PROGRAM MAIN
VAR CONSTANT
	//Constants to set maximum matrix size at compile time
	cMaxRows:INT:=4;
	cMaxCols:INT:=3;
END_VAR
VAR
	//Configure Dispense Matrix [4,3]
	fbDispenseMatrix:FB_Matrix;
	aDispenseMatrixConfig : ARRAY [1..cMaxRows,1..cMaxCols] OF ST_SolenoidConfig;
	bDispMatrixEnable:BOOL;
	bDispMatrixReset:BOOL;
	Disp_st_path : ST_Path;
	bDispFindPath: BOOL;
	bDispPathingSwitch:BOOL;
	nDispenseRows:INT:=4;
	nDispenseCols:INT:=3;
	
	//Configure Inlet Matrix [2,3]
	fbInletMatrix:FB_Matrix;
	aInletMatrixConfig: ARRAY [1..cMaxRows,1..cMaxCols] OF ST_SolenoidConfig;
	bInletMatrixEnable:BOOL;
	bInletMatrixReset:BOOL;
	Inlet_st_path : ST_Path;
	bInletFindPath: BOOL;
	bInletPathingSwitch:BOOL;
	nInletRows:INT:=2;
	nInletCols:INT:=3;
	
	//Configure Filling Matrix [4,3]
	fbFillMatrix:FB_Matrix;
	aFillMatrixConfig : ARRAY [1..cMaxRows,1..cMaxCols] OF ST_SolenoidConfig;
	bFillMatrixEnable:BOOL;
	bFillMatrixReset:BOOL;
	Fill_st_path : ST_Path;
	bFillFindPath: BOOL;
	bFillPathingSwitch:BOOL;
	nFillRows:INT:=4;
	nFillCols:INT:=3;	
	
	//Array of Pressure Transducers
	aPT: ARRAY [1.. GVL_IO.cNumofPT] OF FB_PressureTransducer;
	
	//Standard Config Parameter Struct for Pressure and Temp sensors
	stAnalogCfg : ST_AnalogPressureTemp;
	
	//Initialising Boolean 
	bInitialise:BOOL:=TRUE;
END_VAR

//Run Initialise Method once on first cycle
IF bInitialise THEN
	M_Initalize();
	bInitialise:=FALSE;
END_IF

//Update sensors from IO
M_Sensors();

//Calling FB_MAtrix for each of the three matrices of valves, Dispense, Inlet and FIlling.
fbDispenseMatrix(bDeviceEnable:=bDispMatrixEnable,bDeviceReset:=bDispMatrixReset,
	            aConfig:=aDispenseMatrixConfig,st_path:=Disp_st_path,bSetCurrentPath:=bDispFindPath,
                bPathingOn:=bDispPathingSwitch,nRowSize:=nDispenseRows,nColSize:=nDispenseCols);
				
fbInletMatrix(bDeviceEnable:=bInletMatrixEnable,bDeviceReset:=bInletMatrixReset,aConfig:=aInletMatrixConfig,
	          st_path:=Inlet_st_path,bSetCurrentPath:=bInletFindPath,bPathingOn:=bInletPathingSwitch,
			  nRowSize:=nInletRows,nColSize:=nInletCols);
			  
fbFillMatrix(bDeviceEnable:=bFillMatrixEnable,bDeviceReset:=bFillMatrixReset,aConfig:=aFillMatrixConfig,
	          st_path:=Fill_st_path,bSetCurrentPath:=bFillFindPath,bPathingOn:=bFillPathingSwitch,
			  nRowSize:=nFillRows,nColSize:=nFillCols);

				
//Update the inputs to the matrix functions and pressure sensors from GVLs
M_UpdateFromHMI();

METHOD M_ActuateValves
VAR_INPUT
	rows:INT;
	cols:INT;
END_VAR
END_METHOD

METHOD PUBLIC M_Initalize 
VAR
rows:INT;
cols:INT;
END_VAR

//Configure the pressure sensors
	stAnalogCfg.rWarninglevel:=500;
	stAnalogCfg.rErrorLevel:=525;
	stAnalogCfg.rPressureMinSP:=0;
	stAnalogCfg.rPressureMaxSP:=1000;
	stAnalogCfg.rTemperatureMinSP:=-40;
	stAnalogCfg.rTemperatureMaxSP:=125;
	stAnalogCfg.nRawMin:=0;
	stAnalogCfg.nRawMax:=32767;
//Configure the pressure sensors
FOR rows:=1 TO GVL_IO.cNumofPT DO
    aPT[rows].st_AnalogPressureTempdata:=stAnalogCfg;
	apT[rows].sTag:=GVL_IO.sPTTags[rows];
END_FOR


//Initialise all matrices to be NC and to be un-energised
    FOR  rows:=1 TO cMaxRows DO
       FOR  cols:=1 TO cMaxCols DO
          aDispenseMatrixConfig[rows,cols].NormallyOpen:=FALSE;
		  aInletMatrixConfig[rows,cols].NormallyOpen:=FALSE;
		  aDispenseMatrixConfig[rows,cols].bOpen:=FALSE;
		  aInletMatrixConfig[rows,cols].bOpen:=FALSE;
		  aFillMatrixConfig[rows,cols].NormallyOpen:=FALSE;
		  aFillMatrixConfig[rows,cols].bOpen:=FALSE;
       END_FOR
    END_FOR
END_METHOD

METHOD M_Sensors
VAR
	nsensorNumber:INT;
END_VAR
FOR nsensorNumber:=1 TO GVL_IO.cNumofPT DO
	aPT[nsensorNumber](bDeviceEnable:=GVL_HMI.bEnableSensors,
		               bDeviceReset:=GVL_HMI.bResetSensors,
					   nSensorPressure:=GVL_IO.aPressRaw[nsensorNumber],
					   nSensorTemperature:=GVL_IO.aTempRaw[nsensorNumber],
					   rEngPressure=>GVL_HMI.aPV[nsensorNumber],
					   rEngTemperature=>GVL_HMI.aTV[nsensorNumber],
                       eDeviceState=>GVL_HMI.aSensorErrors[nsensorNumber]);			   
END_FOR
END_METHOD

METHOD M_UpdateDispenseFromHMI
VAR
	rows:INT;
	cols:INT;
END_VAR
//Variables for actuating the Dispense matrix updated from GVL here
bDispMatrixEnable:=GVL_HMI.bDispTurnOnMatrix;
bDispMatrixReset:=GVL_HMI.bDispResetMatrix;
Disp_st_path.endPath:=GVL_HMI.eDispEndOfPath;
Disp_st_path.startPath:=GVL_HMI.eDispStartOfPath;
bDispFindPath:=GVL_HMI.bDispActuatePath;
bDispPathingSwitch:=GVL_HMI.bDispTurnOnPathing;

//Change the display state of the matrix valves on the HMI screen
GVL_HMI.aDispStateofValves:=fbDispenseMatrix.aValveStates;

//Condition to avoid manual control when pathing is on
IF GVL_HMI.bDispTurnOnPathing THEN
	RETURN;
END_IF
FOR rows := 1 TO nDispenseRows DO
       FOR cols := 1 TO nDispenseCols DO
          aDispenseMatrixConfig[rows,cols].bOpen:=GVL_HMI.aDispManualValveSelection[rows,cols];
       END_FOR
END_FOR
END_METHOD

METHOD M_UpdateFillFromHMI
VAR
	rows:INT;
	cols:INT;
END_VAR
//Variables for actuating the filling matrix are updated from GVL here
bFillMatrixEnable:=GVL_HMI.bFillTurnOnMatrix;
bFillMatrixReset:=GVL_HMI.bFillResetMatrix;
bFillFindPath:=GVL_HMI.bFillActuatePath;
bFillPathingSwitch:=GVL_HMI.bFillTurnOnPathing;
Fill_st_path.endPath:=GVL_HMI.eFillEndOfPath;
Fill_st_path.startPath:=GVL_HMI.eFillStartOfPath;

//Change the display state of the matrix valves on the HMI screen
GVL_HMI.aFillStateofValves:=fbFillMatrix.aValveStates;


//Condition to avoid manual control when pathing is on
IF GVL_HMI.bFillTurnOnPathing THEN
	RETURN;
END_IF
FOR rows := 1 TO nFillRows DO
       FOR cols := 1 TO nFillCols DO
          aFillMatrixConfig[rows,cols].bOpen:=GVL_HMI.aFillManualValveSelection[rows,cols];
       END_FOR
END_FOR
END_METHOD

METHOD M_UpdateFromHMI
//Update each matrix Independently
M_UpdateDispenseFromHMI();
M_UpdateInletFromHMI();
M_UpdateFillFromHMI();
END_METHOD

METHOD M_UpdateInletFromHMI
VAR
	rows:INT;
	cols:INT;
END_VAR
//Variables for actuating the inlet matrix are updated from the GVL here
bInletMatrixEnable:=GVL_HMI.bInletTurnOnMatrix;
bInletMatrixReset:=GVL_HMI.bInletResetMatrix;
bInletFindPath:=GVL_HMI.bInletActuatePath;
bInletPathingSwitch:=GVL_HMI.bInbletTurnOnPathing;
Inlet_st_path.endPath:=GVL_HMI.eInletEndOfPath;
Inlet_st_path.startPath:=GVL_HMI.eInletStartOfPath;

//Change the display state of the matrix valves on the HMI screen
GVL_HMI.aInletStateofValves:=fbInletMatrix.aValveStates;

//Condition to avoid manual control when pathing is on
IF GVL_HMI.bInbletTurnOnPathing THEN
	RETURN;
END_IF
FOR rows := 1 TO nInletRows DO
       FOR cols := 1 TO nInletCols DO
          aInletMatrixConfig[rows,cols].bOpen:=GVL_HMI.aInletManualValveSelection[rows,cols];
       END_FOR
END_FOR
END_METHOD

END_PROGRAM

(* stored: Version 1.1.0.1
   POU MAIN: Id {606a3699-021a-464e-b575-9f2f01835131}, SpecialFunc None
   Method M_ActuateValves: Id {05054825-7675-44cb-93b9-5418a0e91680}
   Method M_Initalize: Id {c8c10e44-8587-4199-9743-e05feaa06a39}
   Method M_Sensors: Id {8920a687-dbcd-44ce-acc2-10050478d6e7}
   Method M_UpdateDispenseFromHMI: Id {5551aa22-177e-4a8b-ba12-5a3e1e154657}
   Method M_UpdateFillFromHMI: Id {1f387af1-a8e8-4464-8a9a-5150149a1400}
   Method M_UpdateFromHMI: Id {8779a328-bd71-463f-a457-6702a1e02170}
   Method M_UpdateInletFromHMI: Id {c16b0c66-cb74-42d1-a703-df3168c8abc9} *)
